// TIA Portal project "CLP_PI_6_DT_CERTO" (V15.1)

(* hardware
DEVICE "S7-1200 station_1"  S7-1200 Station
   slot 0: "Rack_0"  S7-1200 Rack  Rack  V1.0
   slot 1: "PLC_1"  CPU 1214C DC/DC/DC  6ES7 214-1AG40-0XB0  V4.2
*)

// ===== PLC "PLC_1"  CPU 1214C DC/DC/DC =====

VAR_GLOBAL   // PLC tag table "Default tag table"
   "ROBO_START_OP" AT %Q0.0 : Bool;
   "ARAME_AVANCA" AT %Q0.2 : Bool;
   "ARAME_RECUA" AT %Q0.3 : Bool;
   "ROBO_END_OP" AT %I0.0 : Bool;
   "MODO_AVANCO" AT %M0.0 : Bool;
   "MODO_RECUO" AT %M0.1 : Bool;
   "DBCP+" AT %MW4 : Int;
   "DBCP-" AT %MW6 : Int;
   "INIT_INSPECT" AT %M0.2 : Bool;
   "MODO_CONFIRMA" AT %M0.3 : Bool;
   "ESTOP_IN" AT %I0.3 : Bool;
   "ESTOP_OUT" AT %Q0.1 : Bool;
   "ESTOP_ROBO_OUT" AT %Q0.4 : Bool;
   "RAMPA_ESTOP" AT %M0.4 : Bool;
   "STARTUP_DELAY" AT %M0.5 : Bool;
END_VAR

DATA_BLOCK "MODBUS DATA"   // DB2
{ S7_Optimized_Access := 'FALSE' }
VERSION : 0.1
   VAR
      REG_MB : Array[0..2] of Int;
      CELL_CONTROL : Array[0..15] of Bool;
   END_VAR
BEGIN
   // CELL_CONTROL[0] : MESA_END_OP
   // CELL_CONTROL[1] : MESA_START_OP
   // CELL_CONTROL[4] : MODO_INSPECAO
   // CELL_CONTROL[3] : ERRO_INSPECAO
   // CELL_CONTROL[2] : INSPECAO_OK
   // REG_MB[0] : SETPOINT_ARAME
   // REG_MB[1] : ARAME_ATUAL
   // CELL_CONTROL[5] : DATA_UPDATE
   // REG_MB[2] : TOL_ARAME
   // CELL_CONTROL[6] : PAINEL_ESTOP
   // CELL_CONTROL[7] : BBB_ESTOP
END_DATA_BLOCK

DATA_BLOCK "MBConfig"   // DB7
{ S7_Optimized_Access := 'TRUE' }
VERSION : 0.1
   VAR
      CONNECT : TCON_IP_v4;
      NDR : Bool;
      DR : Bool;
      ERROR : Bool;
      BUSY : Bool;
      STATE : Word;
   END_VAR
BEGIN
   CONNECT.InterfaceId := 64;
   CONNECT.ID := 1;
   CONNECT.ConnectionType := 11;
   CONNECT.RemoteAddress.ADDR[1] := 192;
   CONNECT.RemoteAddress.ADDR[2] := 168;
   CONNECT.RemoteAddress.ADDR[3] := 0;
   CONNECT.LocalPort := 502;
   CONNECT.RemoteAddress.ADDR[4] := 101;
END_DATA_BLOCK

// folder: System blocks/Program resources

DATA_BLOCK "IEC_Timer_0_DB"   // DB5
{ S7_Optimized_Access := 'TRUE' }
AUTHOR : Simatic
FAMILY : IEC
NAME : IEC_TMR
VERSION : 1.0
// stored: InstanceOfName IEC_TIMER
"IEC_TIMER"
BEGIN
END_DATA_BLOCK

DATA_BLOCK "IEC_Timer_0_DB_1"   // DB6
{ S7_Optimized_Access := 'TRUE' }
AUTHOR : Simatic
FAMILY : IEC
NAME : IEC_TMR
VERSION : 1.0
// stored: InstanceOfName IEC_TIMER
"IEC_TIMER"
BEGIN
END_DATA_BLOCK

DATA_BLOCK "IEC_Timer_0_DB_3"   // DB8
{ S7_Optimized_Access := 'TRUE' }
AUTHOR : Simatic
FAMILY : IEC
NAME : IEC_TMR
VERSION : 1.0
// stored: InstanceOfName IEC_TIMER
"IEC_TIMER"
BEGIN
END_DATA_BLOCK

// folder: (top level)

ORGANIZATION_BLOCK "Main"   // OB1, LAD, ProgramCycle
TITLE = "Main Program Sweep (Cycle)"
{ S7_Optimized_Access := 'TRUE' }
VERSION : 0.1
   VAR_INPUT
      Initial_Call : Bool;   // Initial call of this OB
      Remanence : Bool;   // =True, if remanent data are available
   END_VAR
   VAR_TEMP   // added for the SCL form of the ladder/FBD networks
      _w1 : Bool;
      _w2 : Bool;
      _w3 : Bool;
   END_VAR
BEGIN

REGION Network 1: CICLO DE EMERGÊNCIA
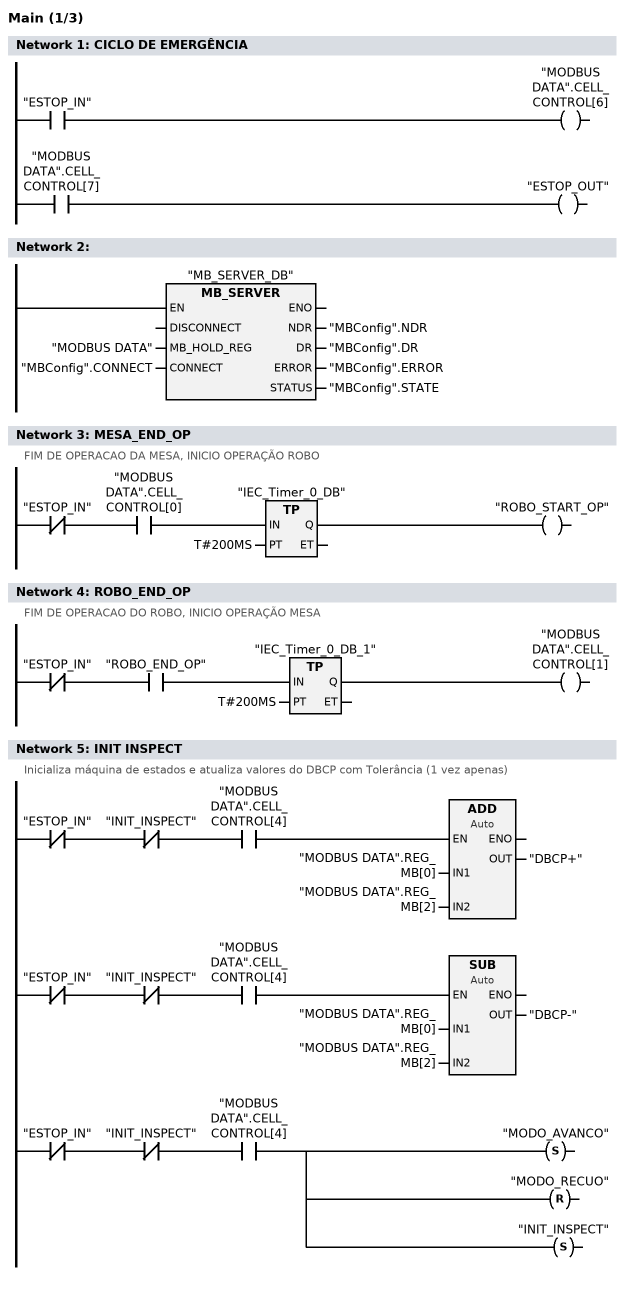
   RUNG wire#powerrail
      Contact( "ESTOP_IN" )
      Coil( "MODBUS DATA".CELL_CONTROL[6] )
   END_RUNG
   RUNG wire#powerrail
      Contact( "MODBUS DATA".CELL_CONTROL[7] )
      Coil( "ESTOP_OUT" )
   END_RUNG
   // the same network as SCL:
   "MODBUS DATA".CELL_CONTROL[6] := "ESTOP_IN";
   "ESTOP_OUT" := "MODBUS DATA".CELL_CONTROL[7];
END_REGION

REGION Network 2
   "MB_SERVER_DB"(MB_HOLD_REG := "MODBUS DATA",   // MB_SERVER
                  CONNECT := "MBConfig".CONNECT,
                  NDR => "MBConfig".NDR,
                  DR => "MBConfig".DR,
                  ERROR => "MBConfig".ERROR,
                  STATUS => "MBConfig".STATE);
END_REGION

REGION Network 3: MESA_END_OP
   // FIM DE OPERACAO DA MESA, INICIO OPERAÇÃO ROBO
   "IEC_Timer_0_DB".TP(IN := NOT "ESTOP_IN" AND "MODBUS DATA".CELL_CONTROL[0], PT := T#200MS);
   "ROBO_START_OP" := "IEC_Timer_0_DB".Q;
END_REGION

REGION Network 4: ROBO_END_OP
   // FIM DE OPERACAO DO ROBO, INICIO OPERAÇÃO MESA
   "IEC_Timer_0_DB_1".TP(IN := NOT "ESTOP_IN" AND "ROBO_END_OP", PT := T#200MS);
   "MODBUS DATA".CELL_CONTROL[1] := "IEC_Timer_0_DB_1".Q;
END_REGION

REGION Network 5: INIT INSPECT
   // Inicializa máquina de estados e atualiza valores do DBCP com Tolerância (1 vez apenas)
   RUNG wire#powerrail
      I_Contact( "ESTOP_IN" )
      I_Contact( "INIT_INSPECT" )
      Contact( "MODBUS DATA".CELL_CONTROL[4] )
      Add(in1 := "MODBUS DATA".REG_MB[0], in2 := "MODBUS DATA".REG_MB[2], out => "DBCP+")
   END_RUNG
   RUNG wire#powerrail
      I_Contact( "ESTOP_IN" )
      I_Contact( "INIT_INSPECT" )
      Contact( "MODBUS DATA".CELL_CONTROL[4] )
      Sub(in1 := "MODBUS DATA".REG_MB[0], in2 := "MODBUS DATA".REG_MB[2], out => "DBCP-")
   END_RUNG
   RUNG wire#powerrail
      I_Contact( "ESTOP_IN" )
      I_Contact( "INIT_INSPECT" )
      Contact( "MODBUS DATA".CELL_CONTROL[4] )
      wire#w1
      S_Coil( "MODO_AVANCO" )
   END_RUNG
   RUNG wire#w1
      R_Coil( "MODO_RECUO" )
   END_RUNG
   RUNG wire#w1
      S_Coil( "INIT_INSPECT" )
   END_RUNG
   // the same network as SCL:
   IF NOT "ESTOP_IN" AND NOT "INIT_INSPECT" AND "MODBUS DATA".CELL_CONTROL[4] THEN
       "DBCP+" := "MODBUS DATA".REG_MB[0] + "MODBUS DATA".REG_MB[2];
       "DBCP-" := "MODBUS DATA".REG_MB[0] - "MODBUS DATA".REG_MB[2];
       "MODO_AVANCO" := TRUE;
       "MODO_RECUO" := FALSE;
       "INIT_INSPECT" := TRUE;
   END_IF;
END_REGION

REGION Network 6: INSPECTION LOGIC
   // Estagio lógico da máquina de estados
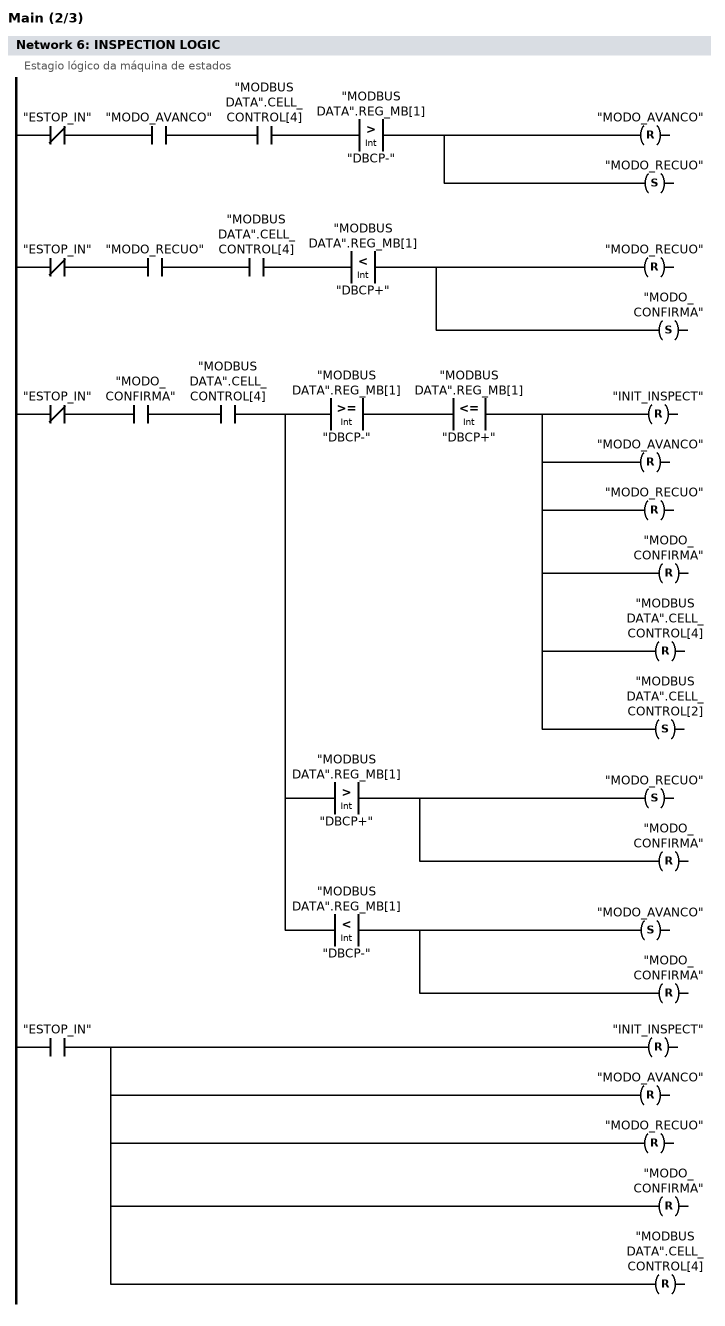
   RUNG wire#powerrail
      I_Contact( "ESTOP_IN" )
      Contact( "MODO_AVANCO" )
      Contact( "MODBUS DATA".CELL_CONTROL[4] )
      { S7_Templates := "SrcType := Int" } GT_Contact(in1 := "MODBUS DATA".REG_MB[1], in2 := "DBCP-")
      wire#w1
      R_Coil( "MODO_AVANCO" )
   END_RUNG
   RUNG wire#w1
      S_Coil( "MODO_RECUO" )
   END_RUNG
   RUNG wire#powerrail
      I_Contact( "ESTOP_IN" )
      Contact( "MODO_RECUO" )
      Contact( "MODBUS DATA".CELL_CONTROL[4] )
      { S7_Templates := "SrcType := Int" } LT_Contact(in1 := "MODBUS DATA".REG_MB[1], in2 := "DBCP+")
      wire#w2
      R_Coil( "MODO_RECUO" )
   END_RUNG
   RUNG wire#w2
      S_Coil( "MODO_CONFIRMA" )
   END_RUNG
   RUNG wire#powerrail
      I_Contact( "ESTOP_IN" )
      Contact( "MODO_CONFIRMA" )
      Contact( "MODBUS DATA".CELL_CONTROL[4] )
      wire#w3
      { S7_Templates := "SrcType := Int" } GE_Contact(in1 := "MODBUS DATA".REG_MB[1], in2 := "DBCP-")
      { S7_Templates := "SrcType := Int" } LE_Contact(in1 := "MODBUS DATA".REG_MB[1], in2 := "DBCP+")
      wire#w4
      R_Coil( "INIT_INSPECT" )
   END_RUNG
   RUNG wire#w4
      R_Coil( "MODO_AVANCO" )
   END_RUNG
   RUNG wire#w4
      R_Coil( "MODO_RECUO" )
   END_RUNG
   RUNG wire#w4
      R_Coil( "MODO_CONFIRMA" )
   END_RUNG
   RUNG wire#w4
      R_Coil( "MODBUS DATA".CELL_CONTROL[4] )
   END_RUNG
   RUNG wire#w4
      S_Coil( "MODBUS DATA".CELL_CONTROL[2] )
   END_RUNG
   RUNG wire#w3
      { S7_Templates := "SrcType := Int" } GT_Contact(in1 := "MODBUS DATA".REG_MB[1], in2 := "DBCP+")
      wire#w5
      S_Coil( "MODO_RECUO" )
   END_RUNG
   RUNG wire#w5
      R_Coil( "MODO_CONFIRMA" )
   END_RUNG
   RUNG wire#w3
      { S7_Templates := "SrcType := Int" } LT_Contact(in1 := "MODBUS DATA".REG_MB[1], in2 := "DBCP-")
      wire#w6
      S_Coil( "MODO_AVANCO" )
   END_RUNG
   RUNG wire#w6
      R_Coil( "MODO_CONFIRMA" )
   END_RUNG
   RUNG wire#powerrail
      Contact( "ESTOP_IN" )
      wire#w7
      R_Coil( "INIT_INSPECT" )
   END_RUNG
   RUNG wire#w7
      R_Coil( "MODO_AVANCO" )
   END_RUNG
   RUNG wire#w7
      R_Coil( "MODO_RECUO" )
   END_RUNG
   RUNG wire#w7
      R_Coil( "MODO_CONFIRMA" )
   END_RUNG
   RUNG wire#w7
      R_Coil( "MODBUS DATA".CELL_CONTROL[4] )
   END_RUNG
   // the same network as SCL:
   #_w1 := NOT "ESTOP_IN" AND "MODO_AVANCO" AND "MODBUS DATA".CELL_CONTROL[4] AND ("MODBUS DATA".REG_MB[1] > "DBCP-");
   IF #_w1 THEN
       "MODO_AVANCO" := FALSE;
       "MODO_RECUO" := TRUE;
   END_IF;
   #_w2 := NOT "ESTOP_IN" AND "MODO_RECUO" AND "MODBUS DATA".CELL_CONTROL[4] AND ("MODBUS DATA".REG_MB[1] < "DBCP+");
   IF #_w2 THEN
       "MODO_RECUO" := FALSE;
       "MODO_CONFIRMA" := TRUE;
   END_IF;
   #_w3 := NOT "ESTOP_IN" AND "MODO_CONFIRMA" AND "MODBUS DATA".CELL_CONTROL[4];
   IF #_w3 AND ("MODBUS DATA".REG_MB[1] >= "DBCP-") AND ("MODBUS DATA".REG_MB[1] <= "DBCP+") THEN
       "INIT_INSPECT" := FALSE;
       "MODO_AVANCO" := FALSE;
       "MODO_RECUO" := FALSE;
       "MODO_CONFIRMA" := FALSE;
       "MODBUS DATA".CELL_CONTROL[4] := FALSE;
       "MODBUS DATA".CELL_CONTROL[2] := TRUE;
   END_IF;
   IF #_w3 AND ("MODBUS DATA".REG_MB[1] > "DBCP+") THEN
       "MODO_RECUO" := TRUE;
       "MODO_CONFIRMA" := FALSE;
   END_IF;
   IF #_w3 AND ("MODBUS DATA".REG_MB[1] < "DBCP-") THEN
       "MODO_AVANCO" := TRUE;
       "MODO_CONFIRMA" := FALSE;
   END_IF;
   IF "ESTOP_IN" THEN
       "INIT_INSPECT" := FALSE;
       "MODO_AVANCO" := FALSE;
       "MODO_RECUO" := FALSE;
       "MODO_CONFIRMA" := FALSE;
       "MODBUS DATA".CELL_CONTROL[4] := FALSE;
   END_IF;
END_REGION

REGION Network 7: INSPECTION ACT
   // ACIONAMNTOS DA MAQUINA DE ESTADO
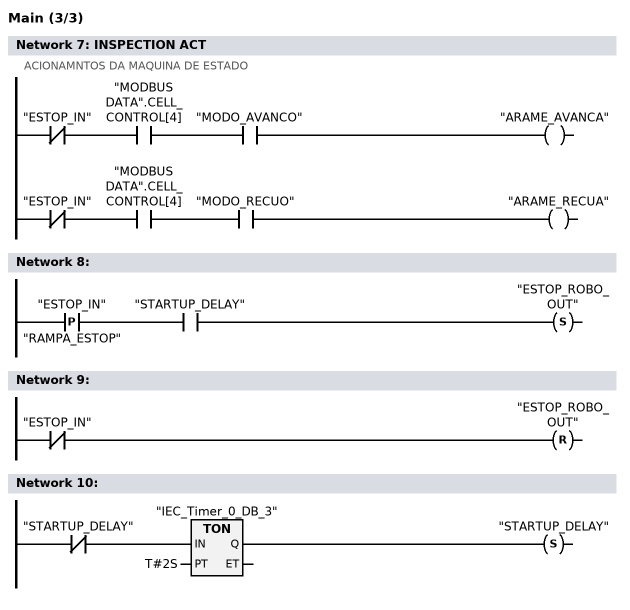
   RUNG wire#powerrail
      I_Contact( "ESTOP_IN" )
      Contact( "MODBUS DATA".CELL_CONTROL[4] )
      Contact( "MODO_AVANCO" )
      Coil( "ARAME_AVANCA" )
   END_RUNG
   RUNG wire#powerrail
      I_Contact( "ESTOP_IN" )
      Contact( "MODBUS DATA".CELL_CONTROL[4] )
      Contact( "MODO_RECUO" )
      Coil( "ARAME_RECUA" )
   END_RUNG
   // the same network as SCL:
   "ARAME_AVANCA" := NOT "ESTOP_IN" AND "MODBUS DATA".CELL_CONTROL[4] AND "MODO_AVANCO";
   "ARAME_RECUA" := NOT "ESTOP_IN" AND "MODBUS DATA".CELL_CONTROL[4] AND "MODO_RECUO";
END_REGION

REGION Network 8
   RUNG wire#powerrail
      P_Contact(operand := "ESTOP_IN", bit := "RAMPA_ESTOP")
      Contact( "STARTUP_DELAY" )
      S_Coil( "ESTOP_ROBO_OUT" )
   END_RUNG
   // the same network as SCL:
   #_w1 := "ESTOP_IN" AND NOT "RAMPA_ESTOP";   // rising edge of "ESTOP_IN"
   "RAMPA_ESTOP" := "ESTOP_IN";
   IF #_w1 AND "STARTUP_DELAY" THEN "ESTOP_ROBO_OUT" := TRUE; END_IF;
END_REGION

REGION Network 9
   RUNG wire#powerrail
      I_Contact( "ESTOP_IN" )
      R_Coil( "ESTOP_ROBO_OUT" )
   END_RUNG
   // the same network as SCL:
   IF NOT "ESTOP_IN" THEN "ESTOP_ROBO_OUT" := FALSE; END_IF;
END_REGION

REGION Network 10
   "IEC_Timer_0_DB_3".TON(IN := NOT "STARTUP_DELAY", PT := T#2S);
   IF "IEC_Timer_0_DB_3".Q THEN "STARTUP_DELAY" := TRUE; END_IF;
END_REGION
END_ORGANIZATION_BLOCK